{attribute 'OPC.UA.DA' := '1'}
TYPE ST_Move_Description :
STRUCT
	accel: LREAL; 
	decel: LREAL; 
	speed: LREAL; 
	max_torque: LREAL; 
END_STRUCT
END_TYPE

(* stored: Version 1.1.0.1, ProductVersion 3.1.4024.13
   DUT ST_Move_Description: Id {85c9793c-c72b-476c-98f8-1c1820b8b7ba} *)
